# EPICS substitutions: stackerApp/Db/stack_0016.substitutions
file "stack_single.template" {
pattern
{ R,        INPR }
{ "\$(R)0", "\$(INPR)0" }
{ "\$(R)1", "\$(INPR)1" }
{ "\$(R)2", "\$(INPR)2" }
{ "\$(R)3", "\$(INPR)3" }
{ "\$(R)4", "\$(INPR)4" }
{ "\$(R)5", "\$(INPR)5" }
{ "\$(R)6", "\$(INPR)6" }
{ "\$(R)7", "\$(INPR)7" }
{ "\$(R)8", "\$(INPR)8" }
{ "\$(R)9", "\$(INPR)9" }
{ "\$(R)A", "\$(INPR)A" }
{ "\$(R)B", "\$(INPR)B" }
{ "\$(R)C", "\$(INPR)C" }
{ "\$(R)D", "\$(INPR)D" }
{ "\$(R)E", "\$(INPR)E" }
{ "\$(R)F", "\$(INPR)F" }
}
